{attribute 'qualified_only'}
{attribute 'strict'}
TYPE E_OPERATION :
(
	Array_Sum 	:= 0,
	Array_Product
);
END_TYPE

(* stored: Version 1.1.0.1, ProductVersion 3.1.4024.12
   EnumerationTextList E_OPERATION: Id {f79f1382-310c-425d-b867-dde06e0e43ee} *)
